ABB RAPID module: CalibData.modx

MODULE CalibData
    PERS tooldata TCPUte:=[TRUE,[[132.071,41.723,98.513],[0.457038964,0.402126676,0.524061687,0.595624774]],[1,[0,0,1],[1,0,0,0],0,0,0]];
    PERS wobjdata Workobject_1:=[FALSE,TRUE,"",[[643.498410119,0,307.999819311],[1,0,0,0]],[[0,0,0],[1,0,0,0]]];
    PERS wobjdata Workobject_2:=[FALSE,TRUE,"",[[676.499807282,78.825773264,368.00041383],[0.633847781,0.633847781,-0.313427807,-0.313427807]],[[0,0,0],[1,0,0,0]]];
ENDMODULE
